(* IEC 61131-3 sources: Industry-PLC-LLM/data/PLCBEAD_repo/PLCBEAD_PLCEmbed-main/PLC-BEAD/Source/GEB/EASTER, 1 file *)

(* ---- EASTER.ST ---- *)
FUNCTION _INT_TO_UDINT:UDINT
	VAR_INPUT
		IN :	INT;
	END_VAR

	_INT_TO_UDINT := DINT_TO_UDINT(INT_TO_DINT(IN));
END_FUNCTION

FUNCTION SET_DATE:UDINT

	VAR_INPUT
		YEAR  :	INT;
		MONTH :	INT;
		DAY  :	INT;
	END_VAR

	VAR
		count :	INT;
	END_VAR

	IF MONTH > 2 THEN
		count := (MONTH - 1) * 30;
		IF MONTH > 7 THEN
			count := count + DWORD_TO_INT(SHR(DINT_TO_DWORD(INT_TO_DINT(MONTH) - INT_TO_DINT(3)),1));
		ELSE
			count := count + DWORD_TO_INT(SHR(DINT_TO_DWORD(INT_TO_DINT(MONTH) - INT_TO_DINT(4)),1));
		END_IF;
		IF SHL(INT_TO_WORD(YEAR),14) = WORD#0 THEN
			count := count + 1;
		END_IF;
	ELSE
		count := (MONTH - 1) * 31;
	END_IF;
	SET_DATE := (_INT_TO_UDINT(count + DAY  - 1) + DWORD_TO_UDINT(SHR(UDINT_TO_DWORD(_INT_TO_UDINT(YEAR) * UDINT#1461 - UDINT#2878169), 2))) * UDINT#86400;

END_FUNCTION

FUNCTION EASTER:UDINT
	VAR_INPUT
		YEAR  :	INT;
	END_VAR

	VAR
		b :	INT;
		c :	INT;
		oDAY  :	INT;
	END_VAR

	b := (204 - 11 * (YEAR  MOD 19)) MOD 30;
	IF b > 27 THEN b := b - 1; END_IF;
	c := (YEAR  + WORD_TO_INT(SHR(INT_TO_WORD(YEAR),2)) + b - 13) MOD 7;
	oDAY  := 28 + b - c;
	IF oDAY  > 33 THEN
		EASTER := SET_DATE(YEAR, 4, oDAY  - 31);
	ELSE
		EASTER := SET_DATE(YEAR, 3, oDAY);
	END_IF;
END_FUNCTION

PROGRAM program0
  VAR
    LocalVar0 : INT;
	LocalOUT  : UDINT;
  END_VAR
  	LocalOUT := EASTER(LocalVar0);
END_PROGRAM
